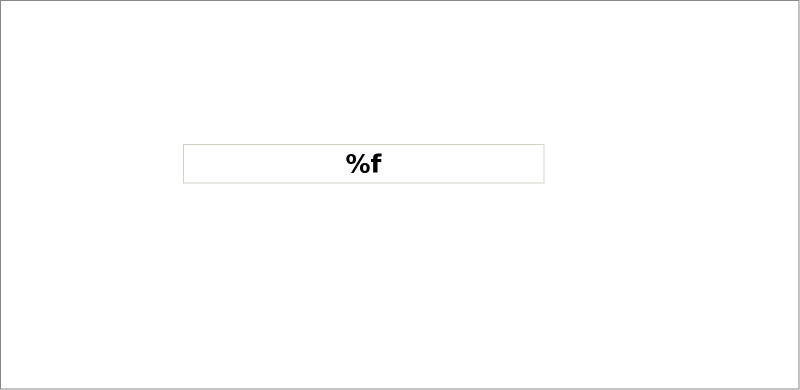
VISUALIZATION VisuEncoderInput  // 800x390
VAR_IN_OUT
	fbManualControler	: FB_ManualController ;
END_VAR
    Textfield (183,144 361x39), "%f", text variable: fbManualControler.pDevEncoder^.nOutPosition
END_VISUALIZATION

(* stored: Version 1.1.0.1, ProductVersion 3.1.4024.9
   Visu VisuEncoderInput: Id {9f88dfcc-1ec2-4c14-8b61-63c3ccc32078} *)
